Staubli VAL3: tooolAndFrame.pgx

program tooolAndFrame()
begin
  for nframe=0 to 9
    frmaster[nframe].trsf=lib:frmaster[nframeSave[nframe]].trsf
    delay(0)
  endFor
  for ntool=0 to 9
    t2[ntool].trsf=lib:t2[ntoolSave[ntool]].trsf
    delay(0)
  endFor
end
